// TwinCAT 3 PLC project DCSv1
// ProgramVersion: 3.1.4023.0
// libraries:
//   Tc2_MC2, * (Beckhoff Automation GmbH)
//   Tc2_MC2_Drive, * (Beckhoff Automation GmbH)
//   Tc2_SerialCom, * (Beckhoff Automation GmbH)
//   Tc2_Standard, * (Beckhoff Automation GmbH)
//   Tc2_System, * (Beckhoff Automation GmbH)
//   Tc2_Utilities, * (Beckhoff Automation GmbH)
//   Tc3_Module, * (Beckhoff Automation GmbH)
// project tree:
//   / ComTask.TcTTO (not stored), PlcTask.TcTTO (not stored)
//   DUTs/ DUT_8BIT.TcDUT
//   GVLs/GVLs/ GVL.TcGVL (not stored), GVL_IO.TcGVL, GVL_PN.TcGVL, GVL_ResearchData.TcGVL, GVL_VAR.TcGVL, ReadMe.TcGVL
//   POUs/FB/ FB_Analog.TcPOU (not stored), F_ScalAnalogOut.TcPOU, F_DecimalData.TcPOU, F_Mapping_REAL.TcPOU, FB_LowpassFilter.TcPOU
//   POUs/ MAIN.TcPOU, P_AP1_Check.TcPOU (not stored), P_ComEL6001.TcPOU (not stored), P_CP1_Check.TcPOU, P_CP1_Enable.TcPOU (not stored), P_Data_Convert.TcPOU (not stored), P_MI1_Curved_Speed.TcPOU (not stored), P_MI1_OnOff.TcPOU (not stored), P_AP1_OnOff.TcPOU (not stored), P_ModeSelector.TcPOU (not stored), P_Outputs_Laptop.TcPOU, P_Outputs_Manual.TcPOU (not stored), P_Set_Research_Data.TcPOU, P_Read_Research_Data.TcPOU, P_SP1_Check.TcPOU, P_SP1_OnOff.TcPOU (not stored)
//   POUs/POUs/ FB_Drive.TcPOU, FB_Mixer1_2.TcPOU (not stored)
// real-time tasks:
//   TASK PlcTask: cycle T#10ms, priority 20, ADS port 350
//   TASK ComTask: cycle T#10ms, priority 21, ADS port 351
// motion (NC):
//   TASK NC-Task 1 SAF: cycle T#2ms, priority 4, ADS port 501
//   TASK NC-Task 1 SVB: cycle T#10ms, priority 8, ADS port 511
//   AXIS Mixer 1 (id 2)
//     General: UnitName=°, UnitFlags=#x00000004
//     Dynamic: Acceleration=7443.34, Deceleration=7443.34, Jerk=22330
//     Velo: RefSearch=49.6222741699219, RefSync=49.6222741699219, SlowManual=248.111370849609, FastManual=1488.66822509766, Fast=4962.22741699219, Maximum=4962.23
//     OtherSettings: AllowMotionCmdToSlave=true
//     encoder EncType=8
//       EncPara: ScaleFactorNumerator=45, ScaleFactorDenominator=1048576, Offset=-131121.7408, Inverse=true, MaxCount=#x007fffff, ReferenceSystem=2
//     drive DrvType=9
//       DrvPara: Inverse=true, MaxCount=#xffffffff, DriveControlDWord=#x00030100
//         Analog: VeloReferenz=5458.45015869141, VeloScale=1.02400649589962, ScaleFactorActTorque=0.1
//         TimeComp: TaskDelayCycles=1
//     controller CtrType=1
//       CtrPara: PriorControlFactor=1
//         Observer: BandWidth=20
//   AXIS Mixer 2 (id 3)
//     General: UnitName=°, UnitFlags=#x00000004
//     Dynamic: Acceleration=7443.34, Deceleration=7443.34, Jerk=22330
//     Velo: RefSearch=49.6222741699219, RefSync=49.6222741699219, SlowManual=248.111370849609, FastManual=1488.66822509766, Fast=4962.22741699219, Maximum=4962.23
//     OtherSettings: AllowMotionCmdToSlave=true
//     encoder EncType=8
//       EncPara: ScaleFactorNumerator=45, ScaleFactorDenominator=1048576, MaxCount=#x007fffff, ReferenceSystem=2
//     drive DrvType=9
//       DrvPara: MaxCount=#xffffffff, DriveControlDWord=#x00030100
//         Analog: VeloReferenz=5458.45015869141, VeloScale=1.02400649589962, ScaleFactorActTorque=0.1
//         TimeComp: TaskDelayCycles=1
//     controller CtrType=1
//       CtrPara: PriorControlFactor=1
//         Observer: BandWidth=20
// I/O:
//   DEVICE Device 1 (EtherCAT), AmsNetId 172.17.147.1.3.1
//     Term 1 (EK1200) [EK1200-5000 EtherCAT Power supply (2A E-Bus)]
//       Term 2 (EL1008) 30K3 [EL1008 8Ch. Dig. Input 24V, 3ms]
//       Term 3 (EL1008) 30K3.1 [EL1008 8Ch. Dig. Input 24V, 3ms]
//       Term 10 (EL1008) new [EL1008 8Ch. Dig. Input 24V, 3ms]
//       Term 4 (EL2008) 30K4 [EL2008 8Ch. Dig. Output 24V, 0.5A]
//       Term 5 (EL2008) 30K5 [EL2008 8Ch. Dig. Output 24V, 0.5A]
//       Term 12 (EL2008) new [EL2008 8Ch. Dig. Output 24V, 0.5A]
//       Term 13 (EL3022) new [EL3022 2Ch. Ana. Input 4-20mA DIFF]
//       Term 14 (EL3202) new [EL3202 2Ch. Ana. Input PT100 (RTD)]
//       Term 16 (EL3202) new pt100 [EL3202 2Ch. Ana. Input PT100 (RTD)]
//       Term 6 (EL3255) 30K5.1 [EL3255 5Ch. potentiometer measurement with sensor supply]
//       Term 7 (EL4134) 30K6 [EL4134 4Ch. Ana. Output -10/+10V, 16bit]
//       Term 8 (EL6001) [EL6001 Interface (RS232)]
//       Term 15 (EL6631-0010) [EL6631-0010 PROFINET IO Device]
//       Term 17 (EL6631) [EL6631 PROFINET IO Controller]
//       Term 9 (EL9011) [EL9011 End Terminal]
//   DEVICE Device 4 (EtherCAT), AmsNetId 172.17.147.1.5.1
//     Drive 11 (AX5206-0000-0213) [AX5206-0000-0213 EtherCAT Drive (SoE, 2 Ch.)]
//   DEVICE Device 1 (EL6631-0010), AmsNetId 5.57.158.168.2.1
//     robotbasicio [ABB Robotics The robot controller's internal PROFINET IO device. 888-3]
//       modules: Term 1 (DAP Module), Term 2 (DI 256 bytes), Term 3 (DO 256 bytes)
// variable links:
//   NC-Task 1 SAF/Axes/Mixer 1 <-> Device 4 (EtherCAT)/Drive 11 (AX5206-0000-0213)
//     Drive/Inputs/In/nDataIn1 <-> AT 1/Following distance
//     Drive/Inputs/In/nDcOutputTime <-> InfoData/DcOutputShift
//     Drive/Inputs/In/nState1 <-> AT 1/Drive status word @bit 8
//     Drive/Inputs/In/nState2 <-> AT 1/Drive status word
//     Drive/Inputs/In/nState4 @bit 1 <-> WcState/InputToggle
//     Drive/Inputs/In/nState4 <-> WcState/WcState
//     Drive/Outputs/Out/nCtrl1 <-> MDT 1/Master control word @bit 8
//     Drive/Outputs/Out/nDataOut1 <-> MDT 1/Position command value
//     Enc/Inputs/In/nDataIn1 <-> AT 1/Position feedback 1 value
//     Enc/Inputs/In/nDcInputTime <-> InfoData/DcInputShift
//     Enc/Inputs/In/nState4 @bit 1 <-> WcState/InputToggle
//     Enc/Inputs/In/nState4 <-> WcState/WcState
//   NC-Task 1 SAF/Axes/Mixer 2 <-> Device 4 (EtherCAT)/Drive 11 (AX5206-0000-0213)
//     Drive/Inputs/In/nDataIn1 <-> AT 2/Following distance
//     Drive/Inputs/In/nDcOutputTime <-> InfoData/DcOutputShift
//     Drive/Inputs/In/nState1 <-> AT 2/Drive status word @bit 8
//     Drive/Inputs/In/nState2 <-> AT 2/Drive status word
//     Drive/Inputs/In/nState4 @bit 1 <-> WcState/InputToggle
//     Drive/Inputs/In/nState4 <-> WcState/WcState
//     Drive/Outputs/Out/nCtrl1 <-> MDT 2/Master control word @bit 8
//     Drive/Outputs/Out/nDataOut1 <-> MDT 2/Position command value
//     Enc/Inputs/In/nDataIn1 <-> AT 2/Position feedback 1 value
//     Enc/Inputs/In/nDcInputTime <-> InfoData/DcInputShift
//     Enc/Inputs/In/nState4 @bit 1 <-> WcState/InputToggle
//     Enc/Inputs/In/nState4 <-> WcState/WcState
//   DCSv1/DCSv1 Instance <-> Device 1 (EL6631-0010)/robotbasicio
//     PlcTask Inputs/GVL_PN.AO_From_ROB <-> API/Term 3 (DO 256 bytes)/Subterm 5 (DO 256 bytes)/Inputs/Output 1
//     PlcTask Inputs/GVL_PN.AO_From_ROB @bit 8 <-> API/Term 3 (DO 256 bytes)/Subterm 5 (DO 256 bytes)/Inputs/Output 2
//     PlcTask Inputs/GVL_PN.DO_From_ROB <-> API/Term 3 (DO 256 bytes)/Subterm 5 (DO 256 bytes)/Inputs/Output 0
//     PlcTask Outputs/GVL_PN.AI_TO_ROB <-> API/Term 2 (DI 256 bytes)/Subterm 4 (DI 256 bytes)/Outputs/Input 1
//     PlcTask Outputs/GVL_PN.AI_TO_ROB @bit 8 <-> API/Term 2 (DI 256 bytes)/Subterm 4 (DI 256 bytes)/Outputs/Input 2
//   DCSv1/DCSv1 Instance <-> Device 1 (EtherCAT)/Term 1 (EK1200)/Term 10 (EL1008) new
//     PlcTask Inputs/GVL_IO.ib_SP1_No_Error <-> Channel 2/Input
//     PlcTask Inputs/GVL_IO.ib_SP1_Ready <-> Channel 1/Input
//   DCSv1/DCSv1 Instance <-> Device 1 (EtherCAT)/Term 1 (EK1200)/Term 13 (EL3022) new
//     PlcTask Inputs/GVL_IO.in_Pressure_Funnel <-> AI Standard Channel 1/Value
//     PlcTask Inputs/GVL_IO.in_Pressure_Pump <-> AI Standard Channel 2/Value
//   DCSv1/DCSv1 Instance <-> Device 1 (EtherCAT)/Term 1 (EK1200)/Term 14 (EL3202) new
//     PlcTask Inputs/GVL_IO.in_Temp_CPump <-> RTD Inputs Channel 2/Value
//     PlcTask Inputs/GVL_IO.in_Temp_CPump_fresh <-> RTD Inputs Channel 1/Value
//   DCSv1/DCSv1 Instance <-> Device 1 (EtherCAT)/Term 1 (EK1200)/Term 16 (EL3202) new pt100
//     PlcTask Inputs/GVL_IO.in_Temp_Funnel_Outlet <-> RTD Inputs Channel 2/Value
//   DCSv1/DCSv1 Instance <-> Device 1 (EtherCAT)/Term 1 (EK1200)/Term 2 (EL1008) 30K3
//     PlcTask Inputs/GVL_IO.ib_AP1_No_Error <-> Channel 6/Input
//     PlcTask Inputs/GVL_IO.ib_AP1_Ready <-> Channel 5/Input
//     PlcTask Inputs/GVL_IO.ib_CC1_Button_Mode_Laptop <-> Channel 8/Input
//     PlcTask Inputs/GVL_IO.ib_CC1_Button_Reset <-> Channel 7/Input
//     PlcTask Inputs/GVL_IO.ib_CC1_Safety_Ready <-> Channel 1/Input
//     PlcTask Inputs/GVL_IO.ib_CP1_Drive_Error <-> Channel 4/Input
//     PlcTask Inputs/GVL_IO.ib_CP1_Ready <-> Channel 3/Input
//     PlcTask Inputs/GVL_IO.ib_CP1_Safety_Grid_Mounted <-> Channel 2/Input
//   DCSv1/DCSv1 Instance <-> Device 1 (EtherCAT)/Term 1 (EK1200)/Term 3 (EL1008) 30K3.1
//     PlcTask Inputs/GVL_IO.ib_AP1_Button_Not_Off <-> Channel 7/Input
//     PlcTask Inputs/GVL_IO.ib_AP1_Button_On <-> Channel 6/Input
//     PlcTask Inputs/GVL_IO.ib_CC1_Button_Mode_Manual <-> Channel 1/Input
//     PlcTask Inputs/GVL_IO.ib_MI1_Button_Not_Off <-> Channel 3/Input
//     PlcTask Inputs/GVL_IO.ib_MI1_Button_On <-> Channel 2/Input
//     PlcTask Inputs/GVL_IO.ib_SP1_Button_Not_Off <-> Channel 5/Input
//     PlcTask Inputs/GVL_IO.ib_SP1_Button_On <-> Channel 4/Input
//   DCSv1/DCSv1 Instance <-> Device 1 (EtherCAT)/Term 1 (EK1200)/Term 4 (EL2008) 30K4
//     PlcTask Outputs/GVL_IO.ob_AP1_Pressure_Ok <-> Channel 7/Output
//     PlcTask Outputs/GVL_IO.ob_AP1_Pulse <-> Channel 8/Output
//     PlcTask Outputs/GVL_IO.ob_AP1_Start <-> Channel 6/Output
//     PlcTask Outputs/GVL_IO.ob_CC1_Safety_Reset <-> Channel 1/Output
//     PlcTask Outputs/GVL_IO.ob_CP1_Backward <-> Channel 5/Output
//     PlcTask Outputs/GVL_IO.ob_CP1_Forward <-> Channel 4/Output
//     PlcTask Outputs/GVL_IO.ob_CP1_Start <-> Channel 3/Output
//     PlcTask Outputs/GVL_IO.ob_CP1_Stop <-> Channel 2/Output
//   DCSv1/DCSv1 Instance <-> Device 1 (EtherCAT)/Term 1 (EK1200)/Term 5 (EL2008) 30K5
//     PlcTask Outputs/GVL_IO.ob_AP1_Not_Empty <-> Channel 1/Output
//     PlcTask Outputs/GVL_IO.ob_AP1_Power_On <-> Channel 2/Output
//     PlcTask Outputs/GVL_IO.ob_SP1_Not_Empty <-> Channel 6/Output
//     PlcTask Outputs/GVL_IO.ob_SP1_Power_On <-> Channel 7/Output
//     PlcTask Outputs/GVL_IO.ob_SP1_Pressure_Ok <-> Channel 4/Output
//     PlcTask Outputs/GVL_IO.ob_SP1_Pulse <-> Channel 5/Output
//     PlcTask Outputs/GVL_IO.ob_SP1_Start <-> Channel 3/Output
//   DCSv1/DCSv1 Instance <-> Device 1 (EtherCAT)/Term 1 (EK1200)/Term 6 (EL3255) 30K5.1
//     PlcTask Inputs/GVL.nInputSpare1 <-> AI Standard Channel 4/Value
//     PlcTask Inputs/GVL.nInputSpare2 <-> AI Standard Channel 5/Value
//     PlcTask Inputs/GVL_IO.in_AP1_Poti_Speed <-> AI Standard Channel 3/Value
//     PlcTask Inputs/GVL_IO.in_MI1_Poti_Speed <-> AI Standard Channel 1/Value
//   DCSv1/DCSv1 Instance <-> Device 1 (EtherCAT)/Term 1 (EK1200)/Term 7 (EL4134) 30K6
//     PlcTask Outputs/GVL_IO.on_AP1_Speed <-> AO Output Channel 2/Analog output
//     PlcTask Outputs/GVL_IO.on_CP1_Speed <-> AO Output Channel 1/Analog output
//     PlcTask Outputs/GVL_IO.on_SP1_Speed <-> AO Output Channel 3/Analog output
//   DCSv1/DCSv1 Instance <-> Device 1 (EtherCAT)/Term 1 (EK1200)/Term 8 (EL6001)
//     ComTask Inputs/GVL.stIn_EL6001/D <-> COM Inputs/Data In 0
//     ComTask Inputs/GVL.stIn_EL6001/D @bit {8..168 step 8} <-> COM Inputs/Data In {1..21}  (21 links)
//     ComTask Inputs/GVL.stIn_EL6001/Status <-> COM Inputs/Status
//     ComTask Outputs/GVL.stOut_EL6001/Ctrl <-> COM Outputs/Ctrl
//     ComTask Outputs/GVL.stOut_EL6001/D <-> COM Outputs/Data Out 0
//     ComTask Outputs/GVL.stOut_EL6001/D @bit {8..168 step 8} <-> COM Outputs/Data Out {1..21}  (21 links)
//   DCSv1/DCSv1 Instance <-> Device 4 (EtherCAT)/Drive 11 (AX5206-0000-0213)
//     PlcTask Inputs/GVL.in_MID1_ActAbsCurrent <-> AT 1/Actual absolute current
//     PlcTask Inputs/GVL.in_MID2_ActAbsCurrent <-> AT 2/Actual absolute current
//     PlcTask Inputs/GVL.in_MID1_ActMotorTemperature <-> AT 1/Motor temperature
//     PlcTask Inputs/GVL.in_MID2_ActMotorTemperature <-> AT 2/Motor temperature
//   DCSv1/DCSv1 Instance <-> NC-Task 1 SAF/Axes/Mixer 1
//     PlcTask Inputs/GVL.Axis_Mixer1.NcToPlc <-> Outputs/ToPlc
//     PlcTask Outputs/GVL.Axis_Mixer1.PlcToNc <-> Inputs/FromPlc
//   DCSv1/DCSv1 Instance <-> NC-Task 1 SAF/Axes/Mixer 2
//     PlcTask Inputs/GVL.Axis_Mixer2.NcToPlc <-> Outputs/ToPlc
//     PlcTask Outputs/GVL.Axis_Mixer2.PlcToNc <-> Inputs/FromPlc

// ---- DUTs/DUT_8BIT.TcDUT
TYPE DUT_8BIT :
STRUCT
	bData:BITARR8;
END_STRUCT
END_TYPE

// ---- GVLs/GVLs/GVL_IO.TcGVL
{attribute 'qualified_only'}
VAR_GLOBAL
//***********************************************************************************
//
// ETH Zürich / Robotic Fabrication Lab
// HIB C 13 / Stefano-Franscini-Platz 1
// CH-8093 Zürich
// 
// ***********************************************************************************
// 
// PROJECT     :  A061 Inline Mixer
// 
// FUNCTION    :  Global Varable In and Outputs
// 
// AUTHOR      :  Fabio Scotto / Philippe Fleischmann
// 
// EMAIL       :  scotto@arch.ethz.ch / fleischmann@arch.ehtz.ch
// 
// Copyright   :  ETH Zürich (CH) 2020
//
// ***********************************************************************************

//
// Inputs

//
// Concrete Controller 1
ib_CC1_Safety_Ready AT %I*: BOOL;
ib_CC1_Button_Mode_Manual AT %I*: BOOL;
ib_CC1_Button_Mode_Laptop AT %I*: BOOL;
//ib_CC1_Button_Mode_Robot AT %I*:BOOL;
//
ib_CC1_Button_Reset AT %I*: BOOL;

//
// Concrete Pump 1
ib_CP1_Drive_Error AT %I*: BOOL;
ib_CP1_Ready AT %I*: BOOL;
ib_CP1_Safety_Grid_Mounted AT %I*: BOOL;
in_CP1_Tube_Pressure_Sensor AT %I*: INT;
in_CP1_Tube_Temperature_Sensor AT %I*: INT;

//
// Peristaltic Pump 1 ( SHOULD BE REMOVE, it is old pump 
// in_PP1_Poti_Speed AT %I*	: INT; 

//
// Accelerator Pump 1
ib_AP1_Button_On AT %I*: BOOL;
ib_AP1_Button_Not_Off AT %I*: BOOL;
ib_AP1_Ready AT %I*: BOOL;
ib_AP1_No_Error AT %I*: BOOL;
in_AP1_Poti_Speed AT %I*	: INT; 

// 
// Superplasticizer Pump 1 (WT 220915)
ib_SP1_Button_On AT %I*: BOOL;
ib_SP1_Button_Not_Off AT %I*: BOOL;
ib_SP1_Ready AT %I*: BOOL;
ib_SP1_No_Error AT %I*: BOOL;
//in_SP1_Poti_Speed AT %I*	: INT; 

//
// Mixer 1
ib_MI1_Button_On AT %I*: BOOL;
ib_MI1_Button_Not_Off AT %I*: BOOL;
in_MI1_Poti_Speed AT %I*	: INT; 

//
// Temperature sensor #WT 20230510
in_Temp_CPump_fresh AT %I*: INT;
in_Temp_Funnel_Outlet AT %I*: INT;
in_Temp_CPump AT %I*: INT;

in_Pressure_Funnel AT %I*: INT;
in_Pressure_Pump AT %I*: INT;

//
// Outputs

//
// Concrete Controller 1
ob_CC1_Safety_Reset AT %Q*: BOOL;

//
// Concrete Pump 1
ob_CP1_Start AT %Q*: BOOL;
ob_CP1_Stop AT %Q*: BOOL;
ob_CP1_Forward AT %Q*: BOOL;
ob_CP1_Backward AT %Q*: BOOL;

on_CP1_Speed AT %Q*: INT;

//
// Accelerator Pump 1
ob_AP1_Power_On AT %Q*: BOOL;
ob_AP1_Start AT %Q*: BOOL;
ob_AP1_Pressure_Ok AT %Q*: BOOL;
ob_AP1_Not_Empty AT %Q*: BOOL;
ob_AP1_Pulse AT %Q*: BOOL;

on_AP1_Speed AT %Q*: INT;

// 
// Superplasticizer Pump 1 (WT 220915)
ob_SP1_Power_On AT %Q*: BOOL;
ob_SP1_Start AT %Q*: BOOL;
ob_SP1_Pressure_Ok AT %Q*: BOOL;
ob_SP1_Not_Empty AT %Q*: BOOL;
ob_SP1_Pulse AT %Q*: BOOL;

on_SP1_Speed AT %Q*: INT;


END_VAR

// ---- GVLs/GVLs/GVL_PN.TcGVL
{attribute 'qualified_only'}
VAR_GLOBAL
	DO_From_ROB AT %I* :BYTE;
	DI_TO_ROB AT %Q* :BYTE;
	DO_From_ROB_2 AT %I* :BYTE;
	DI_TO_ROB_2 AT %Q* :BYTE;
	
	AO_From_ROB AT %I* :WORD;
	AI_TO_ROB AT %Q* :WORD;
END_VAR

// ---- GVLs/GVLs/GVL_ResearchData.TcGVL
{attribute 'qualified_only'}
VAR_GLOBAL
	
//***********************************************************************************
//
// ETH Zürich / Robotic Fabrication Lab
// HIB C 13 / Stefano-Franscini-Platz 1
// CH-8093 Zürich
// 
// ***********************************************************************************
// 
// PROJECT     :  A061 Inline Mixer
// 
// FUNCTION    :  Global Varable to collect all research data
// 
// AUTHOR      :  Seyma Gürel / Philippe Fleischmann / Weiting Chen
// 
// EMAIL       :  scotto@arch.ethz.ch / fleischmann@arch.ehtz.ch
// 
// Copyright   :  ETH Zürich (CH) 2021
//
// ***********************************************************************************


// ***********************************************************************************
// Process inputs
// ***********************************************************************************

// WT ADD 
// Mode 
b_RED_Mode_Manual: BOOL; //Mode
b_RED_Mode_Laptop: BOOL; //Mode


// Temperature and Pressure Sensor
TemperatureAndPressure: STRING := 'TemperatureAndPressure';//***********************************************************

f_RED_Status_Temperature_Funnel_outlet : REAL; // [°C] 
f_RED_Status_Pressure_Funnel_inlet : REAL; // [ bar]

f_RED_Status_Temperature_Concrete_Pump_fresh : REAL; // [°C]
f_RED_Status_Temperature_Concrete_Pump : REAL; // [°C] 
f_RED_Status_Pressure_Concrete_Pump: REAL; // [ bar]


// Power On 
//b_RED_Concrete_Pump_Power_On_Laptop: BOOL;		// NOT USE NOW


//
MIXER: STRING := 'MIXER';//***********************************************************

// Inline Mixer Reactor				
b_RED_Laptop_MI1_Run: BOOL;						// POWER ON *****
f_RED_Control_Speed_by_Laptop:REAL;				// [0 rpm to 120 rpm]
b_RED_Mixer_Curved_Speed_On: BOOL;				// Curved Speed Mode

//
CONCRETE_PUMP: STRING := 'CONCRETE_PUMP';//***************************

// Concrete Pump
b_RED_Concrete_Pump_Forward_On: BOOL;			// Forward ON ******
b_RED_Concrete_Pump_Backward_On: BOOL;			// Forward ON ******
n_RED_Concrete_Pump_Speed: INT;					// **** WRITE VALUE From 0 to 75 ***[rpm] 


b_RED_Concrete_Pump_Check_On: BOOL;				// CHECK MODE ON 
f_RED_Concrete_Pump_Check_Flowrate: REAL; 		// [l/min]
n_RED_Concrete_Pump_Check_Duration_Time: TIME;
f_RED_Concrete_Pump_Density: REAL;				// [g/ml]
f_RED_Concrete_Pump_Check_Mass: REAL;           // [g]

b_RED_Concrete_Pump_Flush_On: BOOL;				// FLUSH MODE ON 
n_RED_Concrete_Pump_Flush_Flowrate: REAL;		// [l/min]

f_RED_Concrete_Pump_Flowrate: REAL; 			// **** WRITE VALUE from _ to 16 [l/min]
f_RED_Concrete_Pump_dosing_volume: REAL;		// calibation 230926 WT


//
Superplasticizer_Pump: STRING := 'Superplasticizer_Pump'; //***************************

// Superplasticizer Pump (WT
b_RED_Superplasticizer_Pump_Power_On_Laptop: BOOL;  // POWER ON 

b_RED_Superplasticizer_Pump_Check_On: BOOL;			// CHECK MODE ON 
n_RED_Superplasticizer_Pump_Check_Flowrate: REAL;
n_RED_Superplasticizer_Pump_Check_Duration: TIME;
f_RED_Superplasticizer_Pump_Density: REAL;          // [g/ml]
f_RED_Superplasticizer_Pump_Mass: REAL;             // [g]

b_RED_Superplasticizer_Pump_Flush_On: BOOL;			// FLUSH MODE ON 
n_RED_Superplasticizer_Pump_Flush_Flowrate: REAL;

n_RED_Superplasticizer_Pump_Max_Flowrate:REAL;
n_RED_Superplasticizer_Pump_Flowrate: REAL;         // **** WRITE VALUE From **** [ml/min]

n_RED_Superplasticizer_Pump_dosing_factor:REAL:=1;

//
ACCELERATION_PUMP: STRING := 'Acceleration_Pump';//***************************

// Accelerator Pump (WT
b_RED_Accelerastor_Pump_Power_On_Laptop: BOOL;  // POWER ON ******

b_RED_Acceleration_Pump_Check_On: BOOL;			// CHECK MODE ON 
n_RED_Acceleration_Pump_Check_Flowrate: REAL;
n_RED_Acceleration_Pump_Check_Duration: TIME;
f_RED_Acceleration_Pump_Density: REAL;          // [g/ml]
f_RED_Acceleration_Pump_Mass: REAL;             // [g]

b_RED_Acceleration_Pump_Flush_On: BOOL;			// FLUSH MODE ON 
n_RED_Acceleration_Pump_Flush_Flowrate: REAL;

n_RED_Acceleration_Pump_Max_Flowrate :REAL;
n_RED_Acceleration_Pump_Flowrate: REAL;         // **** WRITE VALUE From **** [ml/min] 

n_RED_Acceleration_Pump_dosing_factor: REAL:=1;


// ***********************************************************************************
// Process outpus
// ***********************************************************************************

//
PROCESS_OUTPUTS: STRING := 'PROCESS_OUTPUTS';//***********************************************************

// 
// Status mixer
b_RED_Status_On : BOOL;
//f_RED_Status_Speed_Overide : LREAL;
f_RED_Status_Speed_Motor_1 : LREAL;					//[rpm]
f_RED_Status_Speed_Motor_2 : LREAL;					//[rpm]
f_RED_Status_Velo_Motor_1 : LREAL;
f_RED_Status_Velo_Motor_2 :LREAL;

f_RED_Status_Torque_Motor_1 : LREAL;				// [Nm]
f_RED_Status_Torque_Motor_2 : LREAL;				// [Nm]

f_RED_Status_Temperature_Motor_1 : REAL; // [°C] 
f_RED_Status_Temperature_Motor_2 : REAL; // [°C] 


//
// Superplasticizer Pump (WT 220916
//n_RED_Status_Superplasticizer_Pump_Flowrate: INT;          // [ml/min]
f_RED_Status_Superplasticizer_Pump_Max_Flowrate_ml_per_min: REAL;           // [ml/min]

//
// Accelerator Pump
//n_RED_Status_Acceleration_Pump_Flowrate: INT;          // [ml/min]
f_RED_Status_Acceleration_Pump_Max_Flowrate_ml_per_min: REAL;           // [ml/min]

//
//Concrete Pump
f_RED_Status_Concrete_Pump_Max_Flowrate_l_per_min: REAL;           // [l/min]


END_VAR

// ---- GVLs/GVLs/GVL_VAR.TcGVL
{attribute 'qualified_only'}
VAR_GLOBAL
//***********************************************************************************
//
// ETH Zürich / Robotic Fabrication Lab
// HIB C 13 / Stefano-Franscini-Platz 1
// CH-8093 Zürich
// 
// ***********************************************************************************
// 
// PROJECT     :  A061 Inline Mixer
// 
// FUNCTION    :  Global Varable In and Outputs
// 
// AUTHOR      :  Fabio Scotto / Philippe Fleischmann / Weiting Chen
// 
// EMAIL       :  scotto@arch.ethz.ch / fleischmann@arch.ehtz.ch
// 
// Copyright   :  ETH Zürich (CH) 2020
//
// ***********************************************************************************

//
// Concrete Controller 1
b_Mode_Manual : BOOL;
b_Mode_Laptop : BOOL;
b_CC1_Mode_On: BOOL;


//
// Concrete Pump 1

//
// Superplasticizer Pump 1
b_SP1_Run : BOOL;
f_SP1_Override :LREAL;

//
// Accelerator Pump 1
b_AP1_Run : BOOL;
f_AP1_Override : LREAL; 

//
// Mixer 1
b_MI1_ReadToDrive : BOOL;
b_MI1_Run : BOOL;
f_MI1_Override : LREAL; // 0 to 100 [%]
f_MI1_MaxSpeed : LREAL;
f_MI1_ActSpeedM1 : LREAL;
f_MI1_ActSpeedM2 : LREAL;

END_VAR

// ---- GVLs/GVLs/ReadMe.TcGVL
{attribute 'qualified_only'}
VAR_GLOBAL
//***********************************************************************************
//
// ETH Zürich / Robotic Fabrication Lab
// HIB C 13 / Stefano-Franscini-Platz 1
// CH-8093 Zürich
// 
// ***********************************************************************************
// 
// PROJECT     :  A061 Inline Mixer
// 
// FUNCTION    :  Read Me
// 
// AUTHOR      :  Fabio Scotto / Philippe Fleischmann/ Weiting Chen
// 
// EMAIL       :  scotto@arch.ethz.ch / fleischmann@arch.ehtz.ch
// 
// Copyright   :  ETH Zürich (CH) 2020
//
// ***********************************************************************************

//
//Prefix
//ib = Input Bool   / ob = Output Bool
//if = Input float  / of = Output float (REAL, LREAL)
//in = Input numeric/ on = Outplut numerical (INT, Sint, USINT, UNIT, DINT, UDINT, BYTE, WORD, DWORD, LWORD, XINT, UXINT, XWORD) 
//t = Time (TON)



//
//Short Cuts
//CC1 = Concrete Controller 
//AP1 = Accelerator Pump
//CP1 = Concrete Pump
//PP1 = Peristaltic Pump
//MI1 = Mixer
//T1  = Tool 1
//CA1 = Camera 1
//RED = Research Data

END_VAR

// ---- POUs/FB/F_ScalAnalogOut.TcPOU
FUNCTION F_ScalAnalogOut : INT
VAR_INPUT
	n_Input:INT;
	n_InMin:INT;
	n_InMax:INT;
	n_OutMin:INT;
	n_OutMax:INT;

END_VAR
VAR
	f_Input:REAL;
	f_InMin:REAL;
	f_InMax:REAL;
	f_OutMin:REAL;
	f_OutMax:REAL;
	f_DeltaIn:REAL;
	f_DeltaOut:REAL;
END_VAR

//
// Convert integer to real 
f_Input:=INT_TO_REAL(n_Input);
f_InMin:=INT_TO_REAL(n_InMin);
f_InMax:=INT_TO_REAL(n_InMax);
f_OutMin:=INT_TO_REAL(n_OutMin);
f_OutMax:=INT_TO_REAL(n_OutMax);

//
// Check plausibility 

IF f_Input > f_InMax THEN
	f_Input := f_InMax;
END_IF

IF f_InMax = f_InMin THEN	
	//
	// Not plausible output fix value
	F_ScalAnalogOut := 0;
ELSE
	// Check the input data is lager than maximum
	IF f_Input > f_InMax THEN
		f_Input := f_InMax;
	END_IF
	//
	// Plausible calculate output 
	f_DeltaIn:=f_InMax-f_InMin;
	f_DeltaOut:=f_OutMax-f_OutMin;
	F_ScalAnalogOut :=REAL_TO_INT((f_DeltaOut/f_DeltaIn)*(f_Input-f_InMin));	
END_IF

END_FUNCTION

// ---- POUs/FB/F_DecimalData.TcPOU
FUNCTION F_DecimalData : LREAL
VAR_INPUT
	
	//
	data_type : STRING;
	//
	value_input : LREAL;
	
	// decimal places
	n_decimal_digit : INT;
	
	// Round or not
	b_round: BOOL;
	
	// variable for comparison 
	//n_temp_INT : ANY_INT;
	//f_temp_REAL : ANY_REAL;
	//f_temp_LREAL : ANY_REAL;
END_VAR
	
VAR
	value_Output : LREAL;

END_VAR


// This Function is for decimal the data by data type
// only for OUTPUT LREAL and now 

IF data_type = 'REAL' THEN
	
	value_Output:= STRING_TO_REAL(LREAL_TO_FMTSTR(TO_LREAL(value_input), n_decimal_digit, b_round));
	
ELSIF data_type = 'LREAL' THEN
	
	value_Output:= STRING_TO_REAL(LREAL_TO_FMTSTR(value_input, n_decimal_digit, b_round));
	
END_IF

END_FUNCTION

// ---- POUs/FB/F_Mapping_REAL.TcPOU
FUNCTION F_Mapping_REAL : REAL
VAR_INPUT
	f_Input:REAL;
	f_InMin:REAL;
	f_InMax:REAL;
	f_OutMin:REAL;
	f_OutMax:REAL;

END_VAR
VAR
	f_DeltaIn:REAL;
	f_DeltaOut:REAL;
END_VAR

//
// Check plausibility 

IF f_Input > f_InMax THEN
	f_Input := f_InMax;
END_IF

IF f_InMax = f_InMin THEN	
	//
	// Not plausible output fix value
	F_Mapping_REAL := 0;
ELSE
	// Check the input data is lager than maximum
	IF f_Input > f_InMax THEN
		f_Input := f_InMax;
	END_IF
	//
	// Plausible calculate output 
	f_DeltaIn:=f_InMax-f_InMin;
	f_DeltaOut:=f_OutMax-f_OutMin;
	F_Mapping_REAL :=(f_DeltaOut/f_DeltaIn)*(f_Input-f_InMin);	
END_IF

END_FUNCTION

// ---- POUs/FB/FB_LowpassFilter.TcPOU
FUNCTION FB_LowpassFilter : REAL;
VAR_INPUT
	rValueIn	:REAL;
END_VAR
VAR
	rValue_In	:REAL;
	rValue_New	:REAL;	
	rValue_Old	:REAL;
	rFactor	    :REAL := 0.1; // 10% old new value			

END_VAR

//***********************************************************************************
//
// 
// ***********************************************************************************
// 
// PROJECT     :  A061 
// 
// FUNCTION    :  
// 
// AUTHOR      :  Weiting Chen
// 
// EMAIL       :  
// 
// Copyright   :  
//
// ***********************************************************************************

//

rValue_In := rValueIn;

IF rValue_Old = 0 THEN;
	rValue_Old := rValue_In;
	rValue_New := ((1-rFactor)*rValue_Old) + (rFactor*rValue_In);
ELSE
	rValue_Old := rValue_New;
	rValue_New := ((1-rFactor)*rValue_Old) + (rFactor*rValue_In);
END_IF


// Read IO in and out
FB_LowpassFilter := rValue_New;

END_FUNCTION

// ---- POUs/MAIN.TcPOU
PROGRAM MAIN
VAR	

	fb_MC_SetPosition		:FB_SoEAX5000SetPositionOffset;
	pos:LREAL;
	Mixer1_2		: FB_Mixer1_2;
	Analog			: FB_Analog;

	SafetyReset 	: bool;
	b_Enable		: BOOL;
	b_Reset			: BOOL;
	
	Test : MC_ReadStatus;
	
	temp_speed_override: INT;
	
END_VAR

//***********************************************************************************
//
// ETH Zürich / Robotic Fabrication Lab
// HIB C 13 / Stefano-Franscini-Platz 1
// CH-8093 Zürich
// 
// ***********************************************************************************
// 
// PROJECT     :  A061 Inline Mixer
// 
// FUNCTION    :  MAIN Programm
// 
// AUTHOR      :  Mathias Suter 
// 
// EMAIL       :  mathias.suter@solinaut.ch
// 
// Copyright   :  ETH Zürich (CH) 2021
//
// ***********************************************************************************

P_Data_Convert();
//
// Mode selector 
P_ModeSelector();

//
// Set research data 
P_Set_Research_Data();

//WT

//***********************************************************************************
// Superplasticizer Pump
//***********************************************************************************

//
// Superplasticizer Pump 1 Check (220916 WT
P_SP1_Check();

//
// Superplasticizer Pump 1 On/Off
IF NOT GVL_ResearchData.b_RED_Superplasticizer_Pump_Check_On THEN
	//
	// Superplasticizer Pump 1 On/Off
	P_SP1_OnOff();
END_IF

//***********************************************************************************
// Acceleration Pump
//***********************************************************************************

//
// Acceleration Pump 1 check
P_AP1_Check();

//
// Check for Acceleration Pump 1 state
IF NOT GVL_ResearchData.b_RED_Acceleration_Pump_Check_On THEN
	//
	// Acceleration Pump 1 On/Off 
	P_AP1_OnOff();
END_IF


//***********************************************************************************
// Inline Mixer
//***********************************************************************************

//
//
P_MI1_OnOff();

//
// Temporary scaling of the poti and laptop ontrol for the mixer override  (WT 221006
IF GVL_VAR.b_Mode_Laptop THEN
	IF GVL_ResearchData.b_RED_Mixer_Curved_Speed_On THEN
		//
		P_MI1_Curved_Speed();
		//
		temp_speed_override:=F_ScalAnalogOut(
			n_Input:= REAL_TO_INT(P_MI1_Curved_Speed.f_MI1_speed),
			n_InMin:= 0, 
			n_InMax:= 120, 
			n_OutMin:= 0, 
			n_OutMax:= 100);
	ELSE
		temp_speed_override:=F_ScalAnalogOut(
			n_Input:= REAL_TO_INT(GVL_ResearchData.f_RED_Control_Speed_by_Laptop),
			n_InMin:= 0, 
			n_InMax:= 120, 
			n_OutMin:= 0, 
			n_OutMax:= 100);
	END_IF
ELSE
	temp_speed_override:=F_ScalAnalogOut(
		n_Input:= REAL_TO_INT(GVL_IO.in_MI1_Poti_Speed),
		n_InMin:= 0, 
		n_InMax:= 32767, 
		n_OutMin:= 0, 
		n_OutMax:= 100);
END_IF

GVL_VAR.f_MI1_Override:= temp_speed_override;

//
// Mixer 1 + 2
Mixer1_2(
	Mixer1			:= GVL.Axis_Mixer1,
 	Mixer2			:= GVL.Axis_Mixer2,
	f_Velocity		:= GVL_VAR.f_MI1_MaxSpeed,
	b_JogForward	:= FALSE,
	b_JogBackwards	:= GVL_VAR.b_MI1_Run,
 	b_Enable		:= (GVL_VAR.b_Mode_Manual OR GVL_VAR.b_Mode_Laptop) AND GVL_IO.ib_CC1_Safety_Ready,	
 	b_Reset			:= GVL_IO.ib_CC1_Button_Reset,
	f_Override		:= GVL_VAR.f_MI1_Override);	
	(*
	fb_MC_SetPosition(
	Axis			:= GVL.Axis_Mixer2,
	memory			:= 1,
	Feedback		:= 0);*)
	
pos:=GVL.Axis_Mixer2.NcToPlc.ModuloActPos;


// Torque
GVL.f_MID1_ActCurrent:=GVL.in_MID1_ActAbsCurrent * 5.9 / 1000;
GVL.f_MID1_ActTorque:=GVL.f_MID1_ActCurrent * 0.8 * 8; // Torque constante / Gear transaltion # 221214 WT Torque constante to 0.8

GVL.f_MID2_ActCurrent:=gvl.in_MID2_ActAbsCurrent * 5.9 / 1000;
GVL.f_MID2_ActTorque:=GVL.f_MID2_ActCurrent * 0.8 * 8; // Torque constante / Gear transaltion

//
// Write global variable for mixer ready to drive
GVL_VAR.b_MI1_ReadToDrive:=Mixer1_2.b_ReadyToDrive;
	
// 
// Reset 
GVL_IO.ob_CC1_Safety_Reset:=TRUE;
 	
// GVL.bResetSafety	:= safetyReset;


//***********************************************************************************
// Concrete Pump
//***********************************************************************************
P_CP1_Enable();

P_CP1_Check();
// Analog();

//
// Outputs
IF GVL_VAR.b_Mode_Manual THEN
	//	
	P_Outputs_Manual();
	
ELSIF GVL_VAR.b_Mode_Laptop THEN
	//	
	P_Outputs_Laptop();
END_IF

//
// Read researchs data 
P_Read_Research_Data();

END_PROGRAM

// ---- POUs/P_Set_Research_Data.TcPOU
PROGRAM P_Set_Research_Data
VAR
END_VAR

//***********************************************************************************
//
// ETH Zürich / Robotic Fabrication Lab
// HIB C 13 / Stefano-Franscini-Platz 1
// CH-8093 Zürich
// 
// ***********************************************************************************
// 
// PROJECT     :  A061 Inline Mixer
// 
// FUNCTION    :  Set all research data for the process
// 
// AUTHOR      :  Seyma Gürel / Philippe Fleischmann / Weiting Chen
// 
// EMAIL       :  scotto@arch.ethz.ch / fleischmann@arch.ehtz.ch
// 
// Copyright   :  ETH Zürich (CH) 2022
//
// ***********************************************************************************


//***********************************************************************************
// Inline mixer 
//***********************************************************************************

// Updating Mixer 1 max speed
GVL_VAR.f_MI1_MaxSpeed:= 720; // [distance/s] ( equel to 120 rpm, by measurement 221006)



//***********************************************************************************
// Superplasticizer pump 
//***********************************************************************************

//Superplasticizer Pump checking values (WT useing for CAC 240208
GVL_ResearchData.n_RED_Superplasticizer_Pump_Check_Flowrate:=GVL_ResearchData.n_RED_Superplasticizer_Pump_Max_Flowrate/2;             // [ml/min]
GVL_ResearchData.n_RED_Superplasticizer_Pump_Max_Flowrate:=138;				// Calibration number 240208 138 (122ml/min 5018 rev/min(rpm) in VIsco proparam driver) 

GVL_ResearchData.n_RED_Superplasticizer_Pump_Check_Duration:=T#60000MS;     // [ms]
//GVL_ResearchData.f_RED_Superplasticizer_Pump_Density:=1.06;               // [g/cm^3] TODO use for calibration number

GVL_ResearchData.n_RED_Superplasticizer_Pump_Flush_Flowrate:=GVL_ResearchData.f_RED_Status_Superplasticizer_Pump_Max_Flowrate_ml_per_min;	// [ml/min]

//[32767 is equal 10v output and it means maximum setup speed from ViscoTec 3803 rpm]


//***********************************************************************************
// Accelerator pump 1
//***********************************************************************************
//
// Accelerator Pump checking values (WT using for Xseed 240208
GVL_ResearchData.n_RED_Acceleration_Pump_Check_Flowrate:=GVL_ResearchData.n_RED_Acceleration_Pump_Max_Flowrate/2;     		
GVL_ResearchData.n_RED_Acceleration_Pump_Max_Flowrate:=637; 			// Calibration number 240208 (274 ml/min 4800 rev/min(rpm) in VIsco proparam driver) 

GVL_ResearchData.n_RED_Acceleration_Pump_Check_Duration:=T#60000MS;   	// [ms]

//GVL_ResearchData.f_RED_Acceleration_Pump_Density:=1.62;               // [kg/m^3] TODO use for calibration number

GVL_ResearchData.n_RED_Acceleration_Pump_Flush_Flowrate:=GVL_ResearchData.f_RED_Status_Acceleration_Pump_Max_Flowrate_ml_per_min;	// [ml/min]


//[32767 is equal 10v output and it means maximum setup speed from ViscoTec 3517 rpm]
GVL_ResearchData.f_RED_Acceleration_Pump_Mass:= (GVL_ResearchData.n_RED_Acceleration_Pump_Check_Flowrate*
												(TO_REAL(GVL_ResearchData.n_RED_Acceleration_Pump_Check_Duration)/TO_REAL(T#60000MS))*
												GVL_ResearchData.f_RED_Acceleration_Pump_Density);


//***********************************************************************************
// Concrete pump 1
//***********************************************************************************
GVL_ResearchData.f_RED_Concrete_Pump_Check_Flowrate:=2.5;		//[l/min] (1.3 to 3.7)
GVL_ResearchData.n_RED_Concrete_Pump_Check_Duration_Time:=T#15000MS;		// [ms]
GVL_ResearchData.n_RED_Concrete_Pump_Flush_Flowrate:=GVL_ResearchData.f_RED_Status_Concrete_Pump_Max_Flowrate_l_per_min; // [l/min]

//GVL_ResearchData.f_RED_Concrete_Pump_Density:=2.307;		// [kg/m^3]
GVL_ResearchData.f_RED_Concrete_Pump_Check_Mass:= (GVL_ResearchData.f_RED_Concrete_Pump_Check_Flowrate * 1000 *
												(TO_REAL(GVL_ResearchData.n_RED_Concrete_Pump_Check_Duration_Time)/TO_REAL(T#60000MS))*
												GVL_ResearchData.f_RED_Concrete_Pump_Density);

END_PROGRAM

// ---- POUs/P_SP1_Check.TcPOU
PROGRAM P_SP1_Check
VAR_INPUT
	//
	//INT
	n_Step: INT:=0;
END_VAR
VAR
	//
	// BOOL 
	b_Condition: BOOL;
	b_No_Emergency_Stop: BOOL:=TRUE;

	//
	// Timer
	t_SP1_Calibration_Time: TON; 
END_VAR

//***********************************************************************************
//
// ETH Zürich / Robotic Fabrication Lab
// HIB C 13 / Stefano-Franscini-Platz 1
// CH-8093 Zürich
// 
// ***********************************************************************************
// 
// PROJECT     :  A061 
// 
// FUNCTION    :  Step chain for Superplasticizer pump system check
// 
// AUTHOR      :  Weiting Chen / Philippe Fleischmann
// 
// EMAIL       :  
// 
// Copyright   :  
//
// ***********************************************************************************

//
// Ignore emergency stop
b_No_Emergency_Stop:=TRUE;

//
// Initalization
IF n_Step=0 THEN
	//
	// Check condition 
	b_Condition:=TRUE;
	//
	// Do 
	IF b_Condition THEN
		b_Condition:=FALSE;
		n_Step:=10;
	END_IF
END_IF

//
// Wait for activating calibration
IF n_Step=10 THEN
	//
	// Check condition 
	b_Condition:= GVL_ResearchData.b_RED_Superplasticizer_Pump_Check_On;
	//
	// Do
	IF b_Condition THEN
		b_Condition:=FALSE;
		n_Step:=20;
	END_IF
END_IF

//
// Wait for start 
IF n_Step=20 THEN
	//
	// Check condition 
	b_Condition:= GVL_IO.ib_SP1_Ready AND (GVL_IO.ib_SP1_Button_On OR GVL_ResearchData.b_RED_Superplasticizer_Pump_Power_On_Laptop);
	//
	// Do 
	IF b_Condition THEN
		b_Condition:=FALSE;
		n_Step:=30;
	END_IF
END_IF

//
// Run calibration until time is over 
IF n_Step=30 THEN
	//
	// Check condition 
	b_Condition:=t_SP1_Calibration_Time.Q; 
	//
	// Do step
	IF b_Condition THEN
		b_Condition:=FALSE;
		n_Step:=40;
	END_IF
END_IF

//
// Reserve
IF n_Step=40 THEN
	//
	// Check condition 
	b_Condition:=TRUE;
	//
	// Do step
	IF b_Condition AND b_No_Emergency_Stop THEN
		b_Condition:=FALSE;
		n_Step:=50;
	END_IF
END_IF

//
// Return to step 10 
IF n_Step=50 THEN
	//
	// Check condition 
	b_Condition:=TRUE;
	//
	// Do step
	IF b_Condition THEN
		b_Condition:=FALSE;
		//
		// Reset check mode on
		GVL_ResearchData.b_RED_Superplasticizer_Pump_Check_On:=FALSE;
		// Turn Off the pump
		GVL_ResearchData.b_RED_Superplasticizer_Pump_Power_On_Laptop:=FALSE;
		n_Step:=10;
	END_IF
END_IF

// ****************************************
// Timer
// ****************************************
t_SP1_Calibration_Time(
	IN:=n_Step=30,
	PT:=GVL_ResearchData.n_RED_Superplasticizer_Pump_Check_Duration);

// ****************************************
// Reset
// ****************************************
IF NOT GVL_ResearchData.b_RED_Superplasticizer_Pump_Check_On THEN
  //
  // Rest step chain
  n_Step:=0;
END_IF

END_PROGRAM

// ---- POUs/P_CP1_Check.TcPOU
PROGRAM P_CP1_Check
VAR_INPUT
	//
	// INT 
	n_Step: INT := 0;	
END_VAR
VAR
	//
	// BOOL 
	b_Condition: BOOL;
	b_No_Emergency_Stop:BOOL :=TRUE;
	
	//
	// Timer 
	t_CP1_Check_Time: TON;
	//
	t_CP1_Puls_Enable: TON;	
	t_CP1_Puls_Disable: TON;	
	
END_VAR

//***********************************************************************************
//
// ETH Zürich / Robotic Fabrication Lab
// HIB C 13 / Stefano-Franscini-Platz 1
// CH-8093 Zürich
// 
// ***********************************************************************************
// 
// PROJECT     :  A061 
// 
// FUNCTION    :  Step chain for Concrete pump calibration
// 
// AUTHOR      :  Weiting Chen / Philippe Fleischmann
// 
// EMAIL       :  
// 
// Copyright   :  
//
// ***********************************************************************************

// Ignore emergency stop
b_No_Emergency_Stop:=TRUE;

//
// Initalization
IF n_Step=0 THEN
	//
	// Check condition 
	b_Condition:=TRUE;
	//
	// Do step
	IF b_Condition THEN
		b_Condition:=FALSE;
		n_Step:=10;
	END_IF
END_IF

//
// Check grid mounted and no errors and the check mode on 
IF n_Step=10 THEN
	//
	// Check condition 
	b_Condition:= GVL_IO.ib_CP1_Ready AND GVL_IO.ib_CP1_Safety_Grid_Mounted AND NOT GVL_IO.ib_CP1_Drive_Error;
	//
	// Do step
	IF b_Condition AND b_No_Emergency_Stop THEN
		b_Condition:=FALSE;
		n_Step:=20;
	END_IF
END_IF

//
// Send enable to pump and wait for start 
IF n_Step=20 THEN
	//
	// Check condition 
	b_Condition:= GVL_ResearchData.b_RED_Concrete_Pump_Check_On AND GVL_ResearchData.b_RED_Concrete_Pump_Forward_On;
	//
	// Do step
	IF b_Condition AND b_No_Emergency_Stop THEN
		b_Condition:=FALSE;
		n_Step:=25;
	END_IF
END_IF

//
// Pump enabled checking for errors or grid removed
IF n_Step=25 THEN
	//
	// Check condition 
	b_Condition:= t_CP1_Check_Time.Q;
	//
	// Do step
	IF b_Condition THEN
		b_Condition:=FALSE;
		n_Step:=30;
	END_IF
END_IF

//
// Pump enabled checking for errors or grid removed
IF n_Step=30 THEN
	//
	// Check condition 
	b_Condition:= TRUE;
	//
	// Do step
	IF b_Condition THEN
		b_Condition:=FALSE;
		n_Step:=40;
	END_IF
END_IF

//
// 
IF n_Step=40 THEN
	//
	// Check condition 
	b_Condition:=TRUE;
	//
	// Do step
	IF b_Condition AND b_No_Emergency_Stop THEN
		b_Condition:=FALSE;
		n_Step:=50;
	END_IF
END_IF

//
// Return to step 10 
IF n_Step=50 THEN
	//
	// Check condition 
	b_Condition:=TRUE;
	//
	// Do step
	IF b_Condition THEN
		//
		//Reset 
		GVL_ResearchData.b_RED_Concrete_Pump_Check_On:=FALSE;
		GVL_ResearchData.b_RED_Concrete_Pump_Forward_On:=FALSE;
		b_Condition:=FALSE;
		n_Step:=10;
	END_IF
END_IF


// ****************************************
// Timer
// ****************************************
t_CP1_Check_Time(
	IN:=n_Step=25,
	PT:=GVL_ResearchData.n_RED_Concrete_Pump_Check_Duration_Time);

// ****************************************
// Reset
// ****************************************
IF NOT GVL_ResearchData.b_RED_Concrete_Pump_Check_On THEN
  //
  // Rest step chain
  n_Step:=0;
END_IF

END_PROGRAM

// ---- POUs/P_Outputs_Laptop.TcPOU
PROGRAM P_Outputs_Laptop
VAR
	//
	n_temp_speed_SP1: REAL;
	n_temp_speed_AP1: REAL;
	n_temp_speed_MI1: REAL;
	
	n_temp_speed_CP1: REAL;
	n_temp_flowrate_CP1: REAL;
	
	
	// temp data for concrete pump
	n_max_pump_speed: REAL :=75;    // measure value 
	n_target_pump_speed: REAL :=25; // by calibration (7.5L/min)
	n_test_pump_speed: REAL :=50;   // NEW NOTES 230926 current dosing rate is 0.32 L/rev Check real flowrate 50*0.32 = 16L/min
	f_dosing_volume:REAL; 
	
END_VAR

//***********************************************************************************
//
// ETH Zürich / Robotic Fabrication Lab
// HIB C 13 / Stefano-Franscini-Platz 1
// CH-8093 Zürich
// 
// ***********************************************************************************
// 
// PROJECT     :  A061 Digital Casting System
// 
// FUNCTION    :  Outputs Laptop Mode
// 
// AUTHOR      :  Weiting Chen/ Philippe Fleischmann 
// 
// EMAIL       :  chenw@usi.ch
// 
// Copyright   :  USI , ETH Zürich (CH) 2022
//
// ***********************************************************************************


//***********************************************************************************
// Mixer 1
//***********************************************************************************

// pass

//***********************************************************************************
// Superplasticizer pump 1
//***********************************************************************************

//
// Power on
GVL_IO.ob_SP1_Power_On:=GVL_VAR.b_Mode_Laptop;
//
// Pressure is Okay, always set it to True
GVL_IO.ob_SP1_Pressure_Ok:=TRUE;
//
// Bucket is not empty, always set it to true
GVL_IO.ob_SP1_Not_Empty:=TRUE;
//
// Pulse mode is a preset amount,  not in use
GVL_IO.ob_SP1_Pulse:=FALSE;

//
// Start pump
IF		P_SP1_OnOff.n_step= 30 
	OR 	P_SP1_Check.n_Step= 30 
THEN
	//
	// Pump On
	GVL_IO.ob_SP1_Start:=TRUE;
ELSE
	//
	// Pump On
	GVL_IO.ob_SP1_Start:=FALSE;
END_IF

//
// Speeds for Superplastizier pump

IF GVL_ResearchData.b_RED_Superplasticizer_Pump_Flush_On AND P_SP1_OnOff.n_step= 30 THEN
	//
	// Process speed for flushing or filling the pipe
	n_temp_speed_SP1:=GVL_ResearchData.n_RED_Superplasticizer_Pump_Flush_Flowrate;

ELSIF P_SP1_Check.n_Step=20 OR P_SP1_Check.n_Step=30 THEN 	
	//	
	// Check Flowrate for pump
	n_temp_speed_SP1:=GVL_ResearchData.n_RED_Superplasticizer_Pump_Check_Flowrate;
	
ELSE
	//
	// Process speed for pump
	n_temp_speed_SP1:=GVL_ResearchData.n_RED_Superplasticizer_Pump_Flowrate;

END_IF


GVL_IO.on_SP1_Speed:=F_ScalAnalogOut(
	n_Input:= REAL_TO_INT(n_temp_speed_SP1),
	n_InMin:= 0, 
	n_InMax:= REAL_TO_INT(GVL_ResearchData.f_RED_Status_Superplasticizer_Pump_Max_Flowrate_ml_per_min*GVL_ResearchData.n_RED_Superplasticizer_Pump_dosing_factor), 
	n_OutMin:= 0, 
	n_OutMax:= 32767);


//***********************************************************************************
// Accelerator pump 1
//***********************************************************************************

//
// Power on
GVL_IO.ob_AP1_Power_On:=GVL_VAR.b_Mode_Laptop;
//
// Pressure okey always set to true
GVL_IO.ob_AP1_Pressure_Ok:=TRUE;
//
// Bucket not empty always set to true
GVL_IO.ob_AP1_Not_Empty:=TRUE;
//
// Pulse a preset amount not in use
GVL_IO.ob_AP1_Pulse:=FALSE;

//
// Start pump
IF 	   P_AP1_OnOff.n_Step=30 
	OR P_AP1_Check.n_Step=30
THEN
	//
	// Pump on
	GVL_IO.ob_AP1_Start:=TRUE;
ELSE
	//
	// Pump off
	GVL_IO.ob_AP1_Start:=FALSE;
END_IF

//
// Speed for accelerator pump

IF GVL_ResearchData.b_RED_Acceleration_Pump_Flush_On AND P_AP1_OnOff.n_Step=30 THEN
	//
	// Process speed for flushing or filling the pipe
	n_temp_speed_AP1:=GVL_ResearchData.n_RED_Acceleration_Pump_Flush_Flowrate;
ELSIF P_AP1_Check.n_Step=20 OR P_AP1_Check.n_Step=30 THEN
	//	
	// Check Flowrate for pump
	n_temp_speed_AP1:=GVL_ResearchData.n_RED_Acceleration_Pump_Check_Flowrate;
ELSE
	//
	// Process speed for pump
	n_temp_speed_AP1:=GVL_ResearchData.n_RED_Acceleration_Pump_Flowrate;
END_IF

GVL_IO.on_AP1_Speed:=F_ScalAnalogOut(
	n_Input:= REAL_TO_INT(n_temp_speed_AP1),
	n_InMin:= 0, 
	n_InMax:= REAL_TO_INT(GVL_ResearchData.f_RED_Status_Acceleration_Pump_Max_Flowrate_ml_per_min*GVL_ResearchData.n_RED_Acceleration_Pump_dosing_factor), 
	n_OutMin:= 0, 
	n_OutMax:= 32767);


// ***********************************************************************************
// Concrete Pump 1 
// ***********************************************************************************

//
// Start
IF  P_CP1_Enable.n_Step=20 THEN
	GVL_IO.ob_CP1_Start:=TRUE;
ELSE
	GVL_IO.ob_CP1_Start:=FALSE;
END_IF

//
// Stop
IF  P_CP1_Enable.n_Step=40 THEN
	GVL_IO.ob_CP1_Stop:=TRUE;
ELSE
	GVL_IO.ob_CP1_Stop:=FALSE;
END_IF


//
// Forward
GVL_IO.ob_CP1_Forward:=GVL_ResearchData.b_RED_Concrete_Pump_Forward_On;

//
// Backward
GVL_IO.ob_CP1_Backward:=GVL_ResearchData.b_RED_Concrete_Pump_Backward_On;

//
// Concrete pump speed  0 (0V) to 75 rpm (10V)
// Concrete pump max target speed  0 to 25 rpm
// Concrete pump max target Flowrate  0 to 5000 ml/min
// Dosing Volume for Concrete pump is 0.32 L/rev, calibrated 230826 WT 

IF GVL_ResearchData.b_RED_Concrete_Pump_Flush_On THEN
	//
	// Process speed for flushing or filling the pipe
	n_temp_flowrate_CP1:=GVL_ResearchData.f_RED_Status_Concrete_Pump_Max_Flowrate_l_per_min*1000;
ELSIF P_CP1_Check.n_Step=20 OR P_CP1_Check.n_Step=25 THEN
	//	
	// Check Flowrate for pump
	n_temp_flowrate_CP1:=GVL_ResearchData.f_RED_Concrete_Pump_Check_Flowrate*1000;
ELSE
	//
	// Process speed for pump
	n_temp_flowrate_CP1:=GVL_ResearchData.f_RED_Concrete_Pump_Flowrate*1000;
END_IF

//TODO 
GVL_ResearchData.f_RED_Concrete_Pump_dosing_volume:= 0.32;

// temporary remapping  
n_temp_speed_CP1:=F_Mapping_REAL(
	f_Input:= n_temp_flowrate_CP1, 
	f_InMin:= 0, 
	f_InMax:= n_test_pump_speed*GVL_ResearchData.f_RED_Concrete_Pump_dosing_volume*1000,
	f_OutMin:= 0, 
	f_OutMax:= n_test_pump_speed);

// Concrete pump speed  0 (0V) to 75 rpm (10V)
GVL_IO.on_CP1_Speed:=REAL_TO_INT(F_Mapping_REAL(
	f_Input:= n_temp_speed_CP1, 
	f_InMin:= 0, 
	f_InMax:= n_max_pump_speed, 
	f_OutMin:= 0, 
	f_OutMax:= 32767));

END_PROGRAM

// ---- POUs/P_Read_Research_Data.TcPOU
PROGRAM P_Read_Research_Data
VAR
	//
	tempVelo_M1 :LREAL;
	tempVelo_M2 :LREAL;
	
	temp:REAL;

END_VAR

//***********************************************************************************
//
// ETH Zürich / Robotic Fabrication Lab
// HIB C 13 / Stefano-Franscini-Platz 1
// CH-8093 Zürich
// 
// ***********************************************************************************
// 
// PROJECT     :  A061 Inline Mixer
// 
// FUNCTION    :  Read all research data for the process
// 
// AUTHOR      :  Seyma Gürel / Philippe Fleischmann / Weiting Chen
// 
// EMAIL       :  scotto@arch.ethz.ch / fleischmann@arch.ehtz.ch
// 
// Copyright   :  ETH Zürich (CH) 2021
//
// ***********************************************************************************

// 
// Mode [] (WT
GVL_ResearchData.b_RED_Mode_Manual:= GVL_VAR.b_Mode_Manual;
GVL_ResearchData.b_RED_Mode_Laptop:= GVL_VAR.b_Mode_Laptop;

//
// Mixer run []
GVL_ResearchData.b_RED_Status_On:=GVL_ResearchData.b_RED_Laptop_MI1_Run; // SHOULD BE CHANGE 


//
// Mixer 1 speed override [%]
// GVL_ResearchData.f_RED_Status_Speed_Overide:=GVL_VAR.f_MI1_Override;

//
// Mixer 1 current speed []
IF ABS(GVL.Axis_Mixer1.NcToPlc.ActVelo) < 0.5 THEN
	tempVelo_M1:=0;
ELSE
	tempVelo_M1:=ABS(GVL.Axis_Mixer1.NcToPlc.ActVelo);
END_IF
GVL_ResearchData.f_RED_Status_Velo_Motor_1:= tempVelo_M1; 
GVL_ResearchData.f_RED_Status_Speed_Motor_1:= tempVelo_M1/6; 


//
// Mixer 1 current torque []
GVL_ResearchData.f_RED_Status_Torque_Motor_1:= GVL.f_MID1_ActTorque;
//
// Mixer 2 current torque []
GVL_ResearchData.f_RED_Status_Torque_Motor_2:=GVL.f_MID2_ActTorque;

//
// Mixer 1 current motor temperature []
GVL_ResearchData.f_RED_Status_Temperature_Motor_1:=GVL.in_MID1_ActMotorTemperature *0.1; // WT

//
// Mixer 2 current speed []
IF ABS(GVL.Axis_Mixer2.NcToPlc.ActVelo) < 0.5 THEN
	tempVelo_M2:=0;
ELSE
	tempVelo_M2:= ABS(GVL.Axis_Mixer1.NcToPlc.ActVelo);
END_IF
GVL_ResearchData.f_RED_Status_Velo_Motor_2:= tempVelo_M2; 
GVL_ResearchData.f_RED_Status_Speed_Motor_2:= tempVelo_M2/6;

//
// Mixer 1 current motor temperature []
GVL_ResearchData.f_RED_Status_Temperature_Motor_2:=GVL.in_MID2_ActMotorTemperature *0.1; // WT

// Funnel Temperature

GVL_ResearchData.f_RED_Status_Temperature_Concrete_Pump_fresh:= FB_LowpassFilter(INT_TO_REAL(GVL_IO.in_Temp_CPump_fresh)* 0.1);

GVL_ResearchData.f_RED_Status_Temperature_Funnel_outlet:= FB_LowpassFilter(INT_TO_REAL(GVL_IO.in_Temp_Funnel_Outlet) * 0.1); 

GVL_ResearchData.f_RED_Status_Temperature_Concrete_Pump:= FB_LowpassFilter(INT_TO_REAL(GVL_IO.in_Temp_CPump) * 0.1);

//
// Funnel Pressure [0 to 40 bar]
GVL_ResearchData.f_RED_Status_Pressure_Funnel_inlet:= F_Mapping_REAL(
													f_Input:= GVL_IO.in_Pressure_Funnel,
													f_InMin:= 0, 
													f_InMax:= 32767, 
													f_OutMin:= 0, 
													f_OutMax:= 40);
//
// Pump Temperature
GVL_ResearchData.f_RED_Status_Temperature_Concrete_Pump:=GVL_IO.in_Temp_CPump*0;// use for funnel plate temperature !!! 230712
												
// Pump Pressure [0 to 40 bar]
GVL_ResearchData.f_RED_Status_Pressure_Concrete_Pump:= F_Mapping_REAL(
													f_Input:= GVL_IO.in_Pressure_Pump,
													f_InMin:= 0, 
													f_InMax:= 32767, 
													f_OutMin:= 0, 
													f_OutMax:= 40);

//
// Superplasticizer maximum pump flowrate [ml/min]
GVL_ResearchData.f_RED_Status_Superplasticizer_Pump_Max_Flowrate_ml_per_min:=GVL_ResearchData.n_RED_Superplasticizer_Pump_Check_Flowrate*2;

//
// Accelration maximum pump flowrate [ml/min]
GVL_ResearchData.f_RED_Status_Acceleration_Pump_Max_Flowrate_ml_per_min:=GVL_ResearchData.n_RED_Acceleration_Pump_Max_Flowrate;

//
// Concrete pump maximum pump flowrate [ml/min]
GVL_ResearchData.f_RED_Status_Concrete_Pump_Max_Flowrate_l_per_min:=GVL_ResearchData.f_RED_Concrete_Pump_Check_Flowrate*3;

END_PROGRAM

// ---- POUs/POUs/FB_Drive.TcPOU
FUNCTION_BLOCK FB_Drive
VAR_INPUT
	b_Enable				: BOOL;		
	b_Reset					: BOOL;
	f_Override				: LREAL;
	b_JogForward			: BOOL;
	b_JogBackwards			: BOOL;
	b_MoveAbsolute			: BOOL;
	n_MoveAbsoluteDirection	: MC_Direction;
	b_Home					: BOOL;
	f_Velocity				: LREAL;
	f_Acceleration			: LREAL;
	f_Deceleration			: LREAL;
	f_Jerk					: LREAL;
	f_Position				: LREAL;
	
END_VAR
VAR_OUTPUT
	b_PowerActive			: BOOL;
	b_Error					: BOOL;
	n_ErrorID				: UDINT;
	b_MoveAbsoluteDone		: BOOL;
	f_ActVelocity			: LREAL;
	f_ActTorque				: LREAL;
	f_ActPosition			: LREAL;
END_VAR
VAR_IN_OUT
	Axis					: AXIS_REF;
END_VAR
VAR
	fb_MC_Reset				: MC_Reset;
	fb_MC_Power				: MC_Power;
	fb_MC_SetPosition		: FB_SoEAX5000SetPositionOffset;
	fb_MC_Halt				: MC_Halt;
	fb_MC_Jog				: MC_Jog;
	fb_MC_Absolute			: MC_MoveModulo;
END_VAR

//***********************************************************************************
//
// ETH Zürich / Robotic Fabrication Lab
// HIB C 13 / Stefano-Franscini-Platz 1
// CH-8093 Zürich
// 
// ***********************************************************************************
// 
// PROJECT     :  ?? 
// 
// FUNCTION    :  General Function Block for Drives 
// 
// AUTHOR      :  Mathias Suter
// 
// EMAIL       :  mathias.suter@solinaut.ch
// 
// Copyright   :  ETH Zürich (CH) 2021
//
// ***********************************************************************************


//
// Axis Power
fb_MC_Power(
	Axis			:= Axis,    
	Enable          := b_Enable,
    Enable_Positive := b_Enable, 
    Enable_Negative := b_Enable,
    Override        := f_Override);
	
//
// Axis Stop
fb_MC_Halt(
	Axis			:= Axis,
	Execute			:= NOT b_enable,
	Deceleration	:= 1000);
	

//
// Axis Reset	
fb_MC_Reset(
	Axis			:= Axis,    
	Execute         := b_Reset);
	
//
// Axis SetPosition
(*fb_MC_SetPosition(
	Axis			:= Axis,    
	Execute         := b_Home,
	Position		:= f_Position);*)
	
	
fb_MC_SetPosition(
	Axis			:= Axis,    
	Execute         := b_Home,
	memory			:= 1,
	Feedback		:= 0,
	Position		:= f_Position);
	
//
// Axis Jog
fb_MC_Jog(
	Axis			:= Axis,    
	JogForward      := b_JogForward AND fb_MC_Power.Status AND b_Enable,
    JogBackwards 	:= b_JogBackwards AND fb_MC_Power.Status AND b_Enable, 
    Mode 			:= MC_JOGMODE_CONTINOUS,
    Velocity        := f_Velocity,
	Acceleration	:= f_Acceleration,
	Deceleration	:= f_Deceleration,
	Jerk			:= f_Jerk);

//
// Axis Absolute	
fb_MC_Absolute(
	Axis			:= Axis,
	Execute			:= b_MoveAbsolute AND b_Enable,
	Position		:= f_Position,
	Velocity		:= f_Velocity,
	Acceleration	:= f_Acceleration,
	Jerk			:= f_Jerk,
    Direction		:= n_MoveAbsoluteDirection);
	
	
//
// Ouptut Power Active
b_PowerActive := fb_MC_Power.Status;	
	
// Output MoveAbsoluteDone
b_MoveAbsoluteDone := fb_MC_Absolute.Done;

//
// Output Actual Velocity, Torque, Position
f_ActVelocity := Axis.NcToPlc.ActVelo;
f_ActTorque	:= Axis.NcToPlc.ActTorque;
f_ActPosition := Axis.NcToPlc.ModuloActPos;	
		
//
// Output Error
b_Error := fb_MC_Power.Error OR fb_MC_Reset.Error OR fb_MC_SetPosition.Error OR fb_MC_Jog.Error OR fb_MC_Absolute.Error;

//
// Output ErrorID
IF fb_MC_Power.Error THEN
	n_ErrorID := fb_MC_Power.ErrorID;
ELSIF fb_MC_Reset.Error THEN
	n_ErrorID := fb_MC_Reset.ErrorID;
ELSIF fb_MC_SetPosition.Error THEN
	n_ErrorID := fb_MC_SetPosition.ErrorID;
ELSIF fb_MC_Jog.Error THEN
	n_ErrorID := fb_MC_Jog.ErrorID;
ELSIF fb_MC_Absolute.Error THEN
	n_ErrorID := fb_MC_Absolute.ErrorID;
ELSE
	n_ErrorID := 0;	
END_IF;

END_FUNCTION_BLOCK
